{attribute 'qualified_only'}
VAR_GLOBAL
	// Digital Inputs
	bEmgOk 			     AT %I* : BOOL; 
	bStartButton 	     AT %I* : BOOL;
	bStopButton 	     AT %I* : BOOL; 
	bOffSwtich		     AT %I* : BOOL;  
	bManualSwtich	     AT %I* : BOOL; 
	bAutoSwtich			 AT %I* : BOOL; 
	bWinchEnable 		 AT %I* : BOOL; 
	bDisplacementEnable  AT %I* : BOOL;
	
	// Analog Intputs
	fJoyXraw 			 AT %I* : INT; 
	fJoyYraw			 AT %I* : INT; 
	fJoyZraw 			 AT %I* : INT; 
	fPDCVMonitor		 AT %I* : INT; 
	nMoogMonitor		 AT %I* : INT; 
	fYoke				 AT %I* : INT; 
	fPressureWinchA 	 AT %I* : INT; 
	fPressureWinchB 	 AT %I* : INT; 
	fPressureSupply 	 AT %I* : INT; 
	fPressureReturn 	 AT %I* : INT; 
	nWinchEncoderValue	 AT %I* : UDINT; 
	
	// Digital Outputs
	bOpenBrakes 		 AT %Q* : BOOL; 
	bEnablePCDV 		 AT %Q* : BOOL; 
	bWinchValveEnable 	 AT %Q* : BOOL; 
	
	// Analog Outputs
	fWinchPDCVOut 		 AT %Q* : INT := 10000; 
	fWinchValveOut 		 AT %Q* : INT := 16383; 
	
	// New Test
	bTestNew AT %I* : BOOL;
	nTestNew AT %I* : INT;
	
END_VAR

(* stored: Version 1.1.0.1, ProductVersion 3.1.4026.11
   GVL G_IO: Id {2437699e-6b47-4df9-8f46-632e8cfc061f} *)
